ABB RAPID module: Calib_t_Gripper.modx

MODULE Calib_t_Gripper(READONLY)
 LOCAL CONST string dataName := "t_Gripper";
 LOCAL CONST string mechUnitRef := "ROB_1";
 LOCAL CONST string toolRef := "tool0";
 LOCAL CONST robtarget pTCP_Point1 := [[379.0077,122.5044,218.561],[0.05625946,-0.220389,0.9734514,-0.02561104],[0,-1,0,0],[8.999999E+09,8.999999E+09,8.999999E+09,8.999999E+09,8.999999E+09,8.999999E+09]];
 LOCAL CONST robtarget pTCP_Point2 := [[440.3718,-181.6411,218.2788],[0.04652914,-0.992406,0.1011632,0.05226274],[-1,0,-3,0],[8.999999E+09,8.999999E+09,8.999999E+09,8.999999E+09,8.999999E+09,8.999999E+09]];
 LOCAL CONST robtarget pTCP_Point3 := [[503.0711,-45.89736,314.2252],[0.384557,0.6322056,-0.512563,-0.4355584],[-1,-1,-2,0],[8.999999E+09,8.999999E+09,8.999999E+09,8.999999E+09,8.999999E+09,8.999999E+09]];
 !------------------------------------------------------------------------------
 !<auto-generated>
 !This code was generated by a tool.

 !<auto-generated>
 !Changes to this file may cause incorrect behavior and will be lost if
 !the code is regenerated.
 !</auto-generated>
 !------------------------------------------------------------------------------



 ! 28 Jul 2026 12:01:04 by admin from ABB Robotics FlexPendant
 ! Old Value: [TRUE,[[0,1.16,131],[1,0,0,0]],[1,[200,0,0],[1,0,0,0],0,0,0]]
 ! Maxerror, Minerror, Meanerror Values: 0, 0, 0


ENDMODULE
